PROGRAM MAIN
VAR
END_VAR

END_PROGRAM

(* stored: Version 1.1.0.1
   POU MAIN: Id {57ab8f08-f05b-48b4-ac9c-c6301a61b4b2} *)
